{attribute addProperty BoxType "KL8610"}
{attribute addProperty Id "StateAT %I*USINT000Data_InAT %I*INT000CtrlAT %Q*USINT000Data_OutAT %Q*INT000"}
{attribute addProperty CRC "2963801647"}
{attribute addProperty SizeInBites "0"}
{attribute addProperty SizeInBytes "0"}
TYPE KL_B0A8062F :
STRUCT
	{attribute addProperty Name "State"}
	State AT %I* : USINT;
	{attribute addProperty Name "Data_In"}
	Data_In AT %I* : INT;
	{attribute addProperty Name "Ctrl"}
	Ctrl AT %Q* : USINT;
	{attribute addProperty Name "Data_Out"}
	Data_Out AT %Q* : INT;
END_STRUCT
END_TYPE

(* stored: Version 1.2.0.0, ProductVersion 3.1.4024.9
   DUT KL_B0A8062F: Id {71e48536-7f60-46c5-91dc-8a650a5b43bc} *)
